(* IEC 61131-3 sources: Masterarbeit/sigmatek/lasalclass2/PW022_virtualization/Class/_LoadSimulator, 1 file *)

(* ---- _LoadSimulator.st ---- *)
(*!
<Class
	Name               = "_LoadSimulator"
	Revision           = "1.3"
	RealtimeTask       = "true"
	DefRealtime        = "1 ms"
	CyclicTask         = "true"
	DefCyclictime      = "1 ms"
	BackgroundTask     = "true"
	DefBackground      = "always"
	Sigmatek           = "true"
	OSInterface        = "false"
	HighPriority       = "false"
	Automatic          = "false"
	UpdateMode         = "Prescan"
	SharedCommandTable = "true"
	Objectsize         = "(446,120)"
	Comment            = "this class simulates a higher workload&#13;&#10;in each task&#13;&#10;the additional time can be set in the&#13;&#10;provided servers">
	<Channels>
		<Server Name="ActBgTime" Visualized="true" Initialize="false" WriteProtected="false" Retentive="false" Comment="the actual time that is needed for&#13;&#10;background is shown here [µs]&#13;&#10;&#13;&#10;use the read method to get this time&#13;&#10;&#13;&#10;via the write method, the time can &#13;&#10;be reset"/>
		<Server Name="ActCyTime" Visualized="true" Initialize="false" WriteProtected="false" Retentive="false" Comment="the actual time that is needed for&#13;&#10;the cyclic task is shown here [µs]&#13;&#10;&#13;&#10;use the read method to get this time&#13;&#10;&#13;&#10;via the write method, the time can &#13;&#10;be reset"/>
		<Server Name="ActRtTime" Visualized="true" Initialize="false" WriteProtected="false" Retentive="false" Comment="the actual time that is needed for&#13;&#10;the realtime task is shown here [µs]&#13;&#10;&#13;&#10;use the read method to get this time&#13;&#10;&#13;&#10;via the write method, the time can &#13;&#10;be reset"/>
		<Server Name="BgDelay" Visualized="true" Initialize="true" DefValue="200" WriteProtected="false" Retentive="false" Comment="the delay time for the background &#13;&#10;task can be set here [µs]"/>
		<Server Name="ClassSvr" Visualized="false" Initialize="false" WriteProtected="true" Retentive="false"/>
		<Server Name="CyDelay" Visualized="true" Initialize="true" DefValue="100" WriteProtected="false" Retentive="false" Comment="the delay time for the cyclic task &#13;&#10;can be set here [µs]"/>
		<Server Name="MaxBgTime" Visualized="true" Initialize="false" WriteProtected="false" Retentive="false" Comment="the maximal time that is needed for&#13;&#10;background is shown here [µs]&#13;&#10;&#13;&#10;use the read method to get this time&#13;&#10;&#13;&#10;via the write method, the time can &#13;&#10;be reset"/>
		<Server Name="MaxCyTime" Visualized="true" Initialize="false" WriteProtected="false" Retentive="false" Comment="the maximal time that is needed for&#13;&#10;the cyclic task is shown here [µs]&#13;&#10;&#13;&#10;use the read method to get this time&#13;&#10;&#13;&#10;via the write method, the time can &#13;&#10;be reset"/>
		<Server Name="MaxRtTime" Visualized="true" Initialize="false" WriteProtected="false" Retentive="false" Comment="the maximal time that is needed for&#13;&#10;the realtime task is shown here [µs]&#13;&#10;&#13;&#10;use the read method to get this time&#13;&#10;&#13;&#10;via the write method, the time can &#13;&#10;be reset"/>
		<Server Name="RtDelay" Visualized="true" Initialize="true" DefValue="300" WriteProtected="false" Retentive="false" Comment="the delay time for the realtime task &#13;&#10;can be set here [µs]"/>
		<Client Name="EnableBgLoad" Required="false" Internal="false" Comment="if this client gets set to 1, the &#13;&#10;workload of Background Task gets&#13;&#10;started"/>
		<Client Name="EnableCyLoad" Required="false" Internal="false" Comment="if this client gets set to 1, the &#13;&#10;workload of Cyclic Task gets&#13;&#10;started"/>
		<Client Name="EnableRtLoad" Required="false" Internal="false" Comment="if this client gets set to 1, the &#13;&#10;workload of Realtime Task gets&#13;&#10;started"/>
	</Channels>
	<RevDoku>
		<Owner Company="Sigmatek" Author="ObeChr"/>
		<Dokumentation Revision="1.3" Date="2018-04-04" Author="FurLuk" Company="Sigmatek" Description="correction of comments (englisch) and using rules of programming (changing Server names)"/>
		<Dokumentation Revision="1.2" Date="2017-10-19" Author="OC1710198" Company="Sigmatek" Description="Aktuelle Durchlaufzeit + maximale Durchlaufzeit wird nun in der jeweiligen Read-Methode ausgegeben. Dadurch können die Tasks der Klasse entfallen."/>
		<Dokumentation Revision="1.1" Date="2016-09-27" Author="ObeChr" Company="Sigmatek" Description="Simulation der Auslastung kann über Clients aktiviert werden."/>
		<Dokumentation Revision="1.0" Date="2015-02-10" Author="ObeChr" Company="Sigmatek" Description="Erste Version der Klasse zum Belasten der Tasks (Realtime, Cyclic, Background) mit einer definierten Zeit."/>
	</RevDoku>
</Class>
*)
_LoadSimulator : CLASS
  //Servers:
	ClassSvr 	: SvrChCmd_DINT;
	RtDelay 	: SvrCh_UDINT;
	ActRtTime 	: SvrCh_UDINT;
	MaxRtTime 	: SvrCh_UDINT;
	CyDelay 	: SvrCh_UDINT;
	ActCyTime 	: SvrCh_UDINT;
	MaxCyTime 	: SvrCh_UDINT;
	BgDelay 	: SvrCh_UDINT;
	ActBgTime 	: SvrCh_UDINT;
	MaxBgTime 	: SvrCh_UDINT;
  //Clients:
	EnableRtLoad 	: CltCh_DINT;
	EnableCyLoad 	: CltCh_DINT;
	EnableBgLoad 	: CltCh_DINT;
  //Variables:
  //Functions:
				//! <Function Comment="the delay of the cyclic task is done &#13;&#10;here" Name="CyWork"/>
	FUNCTION VIRTUAL GLOBAL CyWork
		VAR_INPUT
			EAX 	: UDINT;
		END_VAR
		VAR_OUTPUT
			state (EAX) 	: UDINT;
		END_VAR;
				//! <Function Comment="the delay of the realtime task is done &#13;&#10;here" Name="RtWork"/>
	FUNCTION VIRTUAL GLOBAL RtWork
		VAR_INPUT
			EAX 	: UDINT;
		END_VAR
		VAR_OUTPUT
			state (EAX) 	: UDINT;
		END_VAR;
				//! <Function Comment="the delay of the background task is&#13;&#10;done here" Name="Background"/>
	FUNCTION VIRTUAL GLOBAL Background
		VAR_INPUT
			EAX 	: UDINT;
		END_VAR
		VAR_OUTPUT
			state (EAX) 	: UDINT;
		END_VAR;

	FUNCTION VIRTUAL GLOBAL ActRtTime::Read
		VAR_OUTPUT
			output (EAX) 	: UDINT;
		END_VAR;

	FUNCTION VIRTUAL GLOBAL ActRtTime::Write
		VAR_INPUT
			input (EAX) 	: UDINT;
		END_VAR
		VAR_OUTPUT
			result (EAX) 	: UDINT;
		END_VAR;

	FUNCTION VIRTUAL GLOBAL MaxRtTime::Read
		VAR_OUTPUT
			output (EAX) 	: UDINT;
		END_VAR;

	FUNCTION VIRTUAL GLOBAL MaxRtTime::Write
		VAR_INPUT
			input (EAX) 	: UDINT;
		END_VAR
		VAR_OUTPUT
			result (EAX) 	: UDINT;
		END_VAR;

	FUNCTION VIRTUAL GLOBAL ActCyTime::Read
		VAR_OUTPUT
			output (EAX) 	: UDINT;
		END_VAR;

	FUNCTION VIRTUAL GLOBAL ActCyTime::Write
		VAR_INPUT
			input (EAX) 	: UDINT;
		END_VAR
		VAR_OUTPUT
			result (EAX) 	: UDINT;
		END_VAR;

	FUNCTION VIRTUAL GLOBAL MaxCyTime::Read
		VAR_OUTPUT
			output (EAX) 	: UDINT;
		END_VAR;

	FUNCTION VIRTUAL GLOBAL MaxCyTime::Write
		VAR_INPUT
			input (EAX) 	: UDINT;
		END_VAR
		VAR_OUTPUT
			result (EAX) 	: UDINT;
		END_VAR;

	FUNCTION VIRTUAL GLOBAL ActBgTime::Read
		VAR_OUTPUT
			output (EAX) 	: UDINT;
		END_VAR;

	FUNCTION VIRTUAL GLOBAL ActBgTime::Write
		VAR_INPUT
			input (EAX) 	: UDINT;
		END_VAR
		VAR_OUTPUT
			result (EAX) 	: UDINT;
		END_VAR;

	FUNCTION VIRTUAL GLOBAL MaxBgTime::Read
		VAR_OUTPUT
			output (EAX) 	: UDINT;
		END_VAR;

	FUNCTION VIRTUAL GLOBAL MaxBgTime::Write
		VAR_INPUT
			input (EAX) 	: UDINT;
		END_VAR
		VAR_OUTPUT
			result (EAX) 	: UDINT;
		END_VAR;
  //Tables:
	FUNCTION @STD
		VAR_OUTPUT
			ret_code	: CONFSTATES;
		END_VAR;
	FUNCTION GLOBAL TAB @CT_;
END_CLASS;

FUNCTION VIRTUAL GLOBAL _LoadSimulator::RtWork
	VAR_INPUT
		EAX 	: UDINT;
	END_VAR
	VAR_OUTPUT
		state (EAX) 	: UDINT;
	END_VAR
  VAR
  	tmpTimeStart  : UDINT;
    tmpTimeEnd    : UDINT;
  END_VAR

  EnableRtLoad := EnableRtLoad.Read();

  // check if the simulation for realtime task is active
  if (EnableRtLoad) then

    // get start time of delay
    tmpTimeStart  := OS_READMICROSEC();
    tmpTimeEnd    := tmpTimeStart;

    // wait until delay time has passed
    while ((tmpTimeEnd - tmpTimeStart) < RtDelay) do

      // get the actual time for comparing
      tmpTimeEnd := OS_READMICROSEC();

    end_while;

  end_if;

	state := READY;

END_FUNCTION

FUNCTION VIRTUAL GLOBAL _LoadSimulator::CyWork
	VAR_INPUT
		EAX 	: UDINT;
	END_VAR
	VAR_OUTPUT
		state (EAX) 	: UDINT;
	END_VAR
  VAR
  	tmpTimeStart  : UDINT;
    tmpTimeEnd    : UDINT;
  END_VAR

  EnableCyLoad := EnableCyLoad.Read();

  // check if the simulation for cyclic task is active
  if (EnableCyLoad) then

    // get start time of delay
    tmpTimeStart  := OS_READMICROSEC();
    tmpTimeEnd    := tmpTimeStart;

    // wait until delay time has passed
    while ((tmpTimeEnd - tmpTimeStart) < CyDelay) do

      // get actual time for comparing
      tmpTimeEnd := OS_READMICROSEC();

    end_while;

  end_if;

	state := READY;

END_FUNCTION

FUNCTION VIRTUAL GLOBAL _LoadSimulator::Background
	VAR_INPUT
		EAX 	: UDINT;
	END_VAR
	VAR_OUTPUT
		state (EAX) 	: UDINT;
	END_VAR
  VAR
  	tmpTimeStart  : UDINT;
    tmpTimeEnd    : UDINT;
  END_VAR

  EnableBgLoad := EnableBgLoad.Read();

  // check if the simulation for background task is active
  if (EnableBgLoad) then

    // get start time of delay
    tmpTimeStart  := OS_READMICROSEC();
    tmpTimeEnd    := tmpTimeStart;

    // wait until delay time has passed
    while ((tmpTimeEnd - tmpTimeStart) < BgDelay) do

      // get actual time for comparing
      tmpTimeEnd := OS_READMICROSEC();

    end_while;

  end_if;

	state := READY;

END_FUNCTION

FUNCTION VIRTUAL GLOBAL _LoadSimulator::ActRtTime::Write
	VAR_INPUT
		input (EAX) 	: UDINT;
	END_VAR
	VAR_OUTPUT
		result (EAX) 	: UDINT;
	END_VAR

  // reset actual time
  _RealAverageTime := 0;

	result := input;

END_FUNCTION

FUNCTION VIRTUAL GLOBAL _LoadSimulator::MaxRtTime::Write
	VAR_INPUT
		input (EAX) 	: UDINT;
	END_VAR
	VAR_OUTPUT
		result (EAX) 	: UDINT;
	END_VAR

  // reset maximal time
  _RealMaximumTime := 0;

	result := input;

END_FUNCTION

FUNCTION VIRTUAL GLOBAL _LoadSimulator::ActCyTime::Write
	VAR_INPUT
		input (EAX) 	: UDINT;
	END_VAR
	VAR_OUTPUT
		result (EAX) 	: UDINT;
	END_VAR

  // reset actual time
  _CyclicAverageTime := 0;

	result := input;

END_FUNCTION

FUNCTION VIRTUAL GLOBAL _LoadSimulator::MaxCyTime::Write
	VAR_INPUT
		input (EAX) 	: UDINT;
	END_VAR
	VAR_OUTPUT
		result (EAX) 	: UDINT;
	END_VAR

  // reset maximal time
  _CyclicMaximumTime := 0;

	result := input;

END_FUNCTION

FUNCTION VIRTUAL GLOBAL _LoadSimulator::ActBgTime::Write
	VAR_INPUT
		input (EAX) 	: UDINT;
	END_VAR
	VAR_OUTPUT
		result (EAX) 	: UDINT;
	END_VAR

  // reset actual time
  _BackgroundAverageTime := 0;

	result := input;

END_FUNCTION

FUNCTION VIRTUAL GLOBAL _LoadSimulator::MaxBgTime::Write
	VAR_INPUT
		input (EAX) 	: UDINT;
	END_VAR
	VAR_OUTPUT
		result (EAX) 	: UDINT;
	END_VAR

  // reset maximal time
  _BackgroundMaximumTime := 0;

	result := input;

END_FUNCTION

FUNCTION VIRTUAL GLOBAL _LoadSimulator::ActRtTime::Read
	VAR_OUTPUT
		output (EAX) 	: UDINT;
	END_VAR

  ActRtTime := _RealAverageTime;
	output := ActRtTime;

END_FUNCTION

FUNCTION VIRTUAL GLOBAL _LoadSimulator::MaxRtTime::Read
	VAR_OUTPUT
		output (EAX) 	: UDINT;
	END_VAR

  MaxRtTime := _RealMaximumTime;
	output := MaxRtTime;

END_FUNCTION

FUNCTION VIRTUAL GLOBAL _LoadSimulator::ActCyTime::Read
	VAR_OUTPUT
		output (EAX) 	: UDINT;
	END_VAR

  ActCyTime := _CyclicAverageTime;
	output := ActCyTime;

END_FUNCTION

FUNCTION VIRTUAL GLOBAL _LoadSimulator::MaxCyTime::Read
	VAR_OUTPUT
		output (EAX) 	: UDINT;
	END_VAR

  MaxCyTime := _CyclicMaximumTime;
	output := MaxCyTime;

END_FUNCTION

FUNCTION VIRTUAL GLOBAL _LoadSimulator::ActBgTime::Read
	VAR_OUTPUT
		output (EAX) 	: UDINT;
	END_VAR

  ActBgTime := _BackgroundAverageTime;
	output := ActBgTime;

END_FUNCTION

FUNCTION VIRTUAL GLOBAL _LoadSimulator::MaxBgTime::Read
	VAR_OUTPUT
		output (EAX) 	: UDINT;
	END_VAR

  MaxBgTime := _BackgroundMaximumTime;
	output := MaxBgTime;

END_FUNCTION
